// TIA Portal V20 export
TYPE "LWONIK_typeOperationMode"
// stored: Access Published
   STRUCT
      auto : Bool;   // Auto Mode
      manual : Bool;   // Manual Mode
      home : Bool;   // Auto Ready Start
      reset : Bool;   // Safety Reset
      enable : Bool;   // OP_Enable
   END_STRUCT;
END_TYPE
